FUNCTION_BLOCK FB_ModeSelector
VAR_INPUT
	bControlBox : BOOL;
END_VAR
VAR_OUTPUT
END_VAR
VAR
	fbMode : FB_ModeVisualization;
END_VAR

IF NOT(bControlBox) THEN
	IF NOT(G_VB.bOn) THEN
		fbMode.Off(TRUE);
		fbMode.Manual(FALSE);
		fbMode.Auto(FALSE);
	ELSIF G_VB.bOn AND NOT(G_VB.bAuto) THEN
		fbMode.Off(FALSE);
		fbMode.Manual(TRUE);
		fbMode.Auto(FALSE);
	ELSIF G_VB.bOn AND G_VB.bAuto THEN
		fbMode.Off(FALSE);
		fbMode.Manual(FALSE);
		fbMode.Auto(TRUE);
	ELSE
		fbMode.Off(FALSE);
		fbMode.Manual(FALSE);
		fbMode.Auto(FALSE);
	END_IF
END_IF

END_FUNCTION_BLOCK

(* stored: Version 1.1.0.1, ProductVersion 3.1.4024.12
   POU FB_ModeSelector: Id {dc4d674e-38ac-46d6-a68e-c41c72f8ff42}, SpecialFunc None *)
